PROGRAM CurrentBPUpdate
VAR
END_VAR

END_PROGRAM

(* stored: Version 1.1.0.1, ProductVersion 3.1.4022.18
   POU CurrentBPUpdate: Id {99ba6aac-1727-45f0-bf15-66d5904d8d8f}, SpecialFunc None *)
